(* Logix 5000 project; controller SX_V040001_C001 vendor 1 type 14 code 77 rev 16.23; software revision 16.04; part 21 of 35 *)
(* tags used below, declared in another part *)
   ALL_KINDS : INT[90];
   Basic : INT;
   G_DInput : DINT[3];
   G_DOutput : DINT[3];
   METERING : INT[44];
   METERING_PULSE : DINT[14];
   NOTDOS : INT[6];
   PARAMETER : INT[501];
(* MainProgram, continued *)

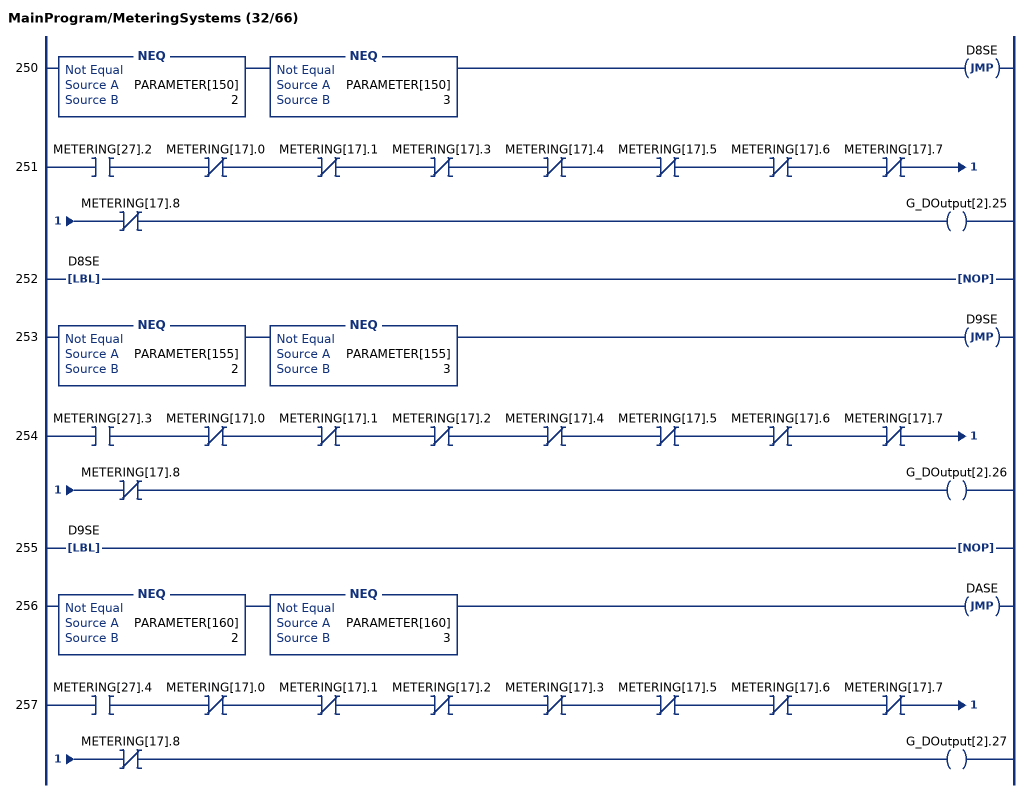
   [picture p456: MainProgram/MeteringSystems rungs 250-257]
   250: NEQ(PARAMETER[150],2)NEQ(PARAMETER[150],3)JMP(D8SE);
   251: XIC(METERING[27].2)XIO(METERING[17].0)XIO(METERING[17].1)XIO(METERING[17].3)XIO(METERING[17].4)XIO(METERING[17].5)XIO(METERING[17].6)XIO(METERING[17].7)XIO(METERING[17].8)OTE(G_DOutput[2].25);
   252: LBL(D8SE)NOP();
   253: NEQ(PARAMETER[155],2)NEQ(PARAMETER[155],3)JMP(D9SE);
   254: XIC(METERING[27].3)XIO(METERING[17].0)XIO(METERING[17].1)XIO(METERING[17].2)XIO(METERING[17].4)XIO(METERING[17].5)XIO(METERING[17].6)XIO(METERING[17].7)XIO(METERING[17].8)OTE(G_DOutput[2].26);
   255: LBL(D9SE)NOP();
   256: NEQ(PARAMETER[160],2)NEQ(PARAMETER[160],3)JMP(DASE);
   257: XIC(METERING[27].4)XIO(METERING[17].0)XIO(METERING[17].1)XIO(METERING[17].2)XIO(METERING[17].3)XIO(METERING[17].5)XIO(METERING[17].6)XIO(METERING[17].7)XIO(METERING[17].8)OTE(G_DOutput[2].27);
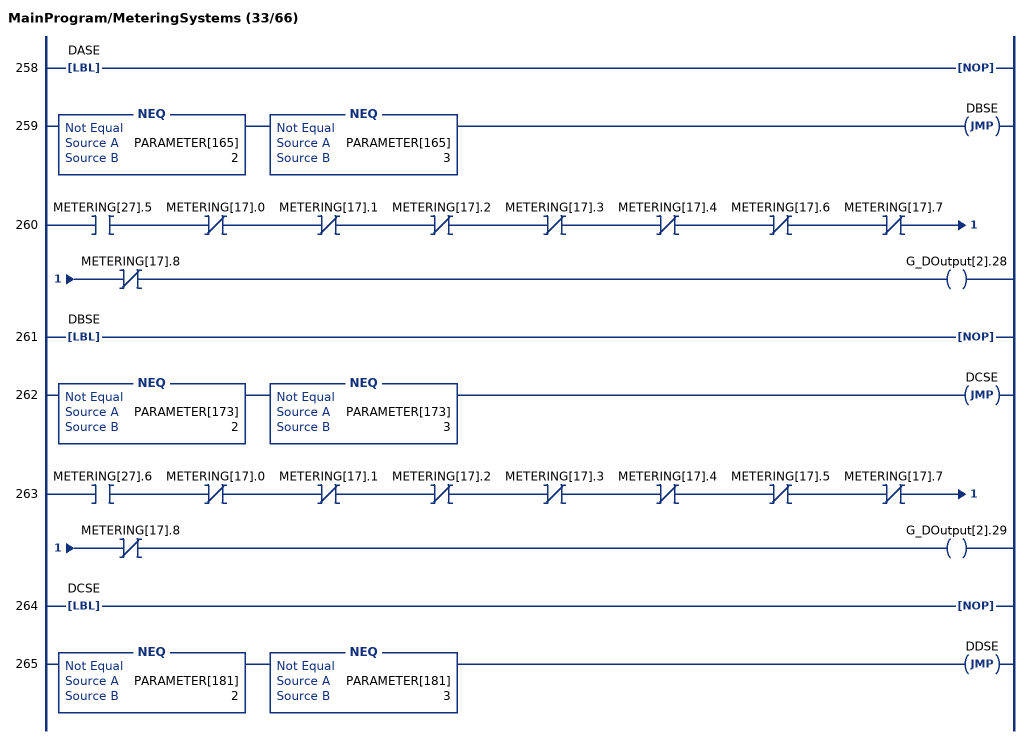
   258: LBL(DASE)NOP();
   259: NEQ(PARAMETER[165],2)NEQ(PARAMETER[165],3)JMP(DBSE);
   260: XIC(METERING[27].5)XIO(METERING[17].0)XIO(METERING[17].1)XIO(METERING[17].2)XIO(METERING[17].3)XIO(METERING[17].4)XIO(METERING[17].6)XIO(METERING[17].7)XIO(METERING[17].8)OTE(G_DOutput[2].28);
   261: LBL(DBSE)NOP();
   262: NEQ(PARAMETER[173],2)NEQ(PARAMETER[173],3)JMP(DCSE);
   263: XIC(METERING[27].6)XIO(METERING[17].0)XIO(METERING[17].1)XIO(METERING[17].2)XIO(METERING[17].3)XIO(METERING[17].4)XIO(METERING[17].5)XIO(METERING[17].7)XIO(METERING[17].8)OTE(G_DOutput[2].29);
   264: LBL(DCSE)NOP();
   265: NEQ(PARAMETER[181],2)NEQ(PARAMETER[181],3)JMP(DDSE);
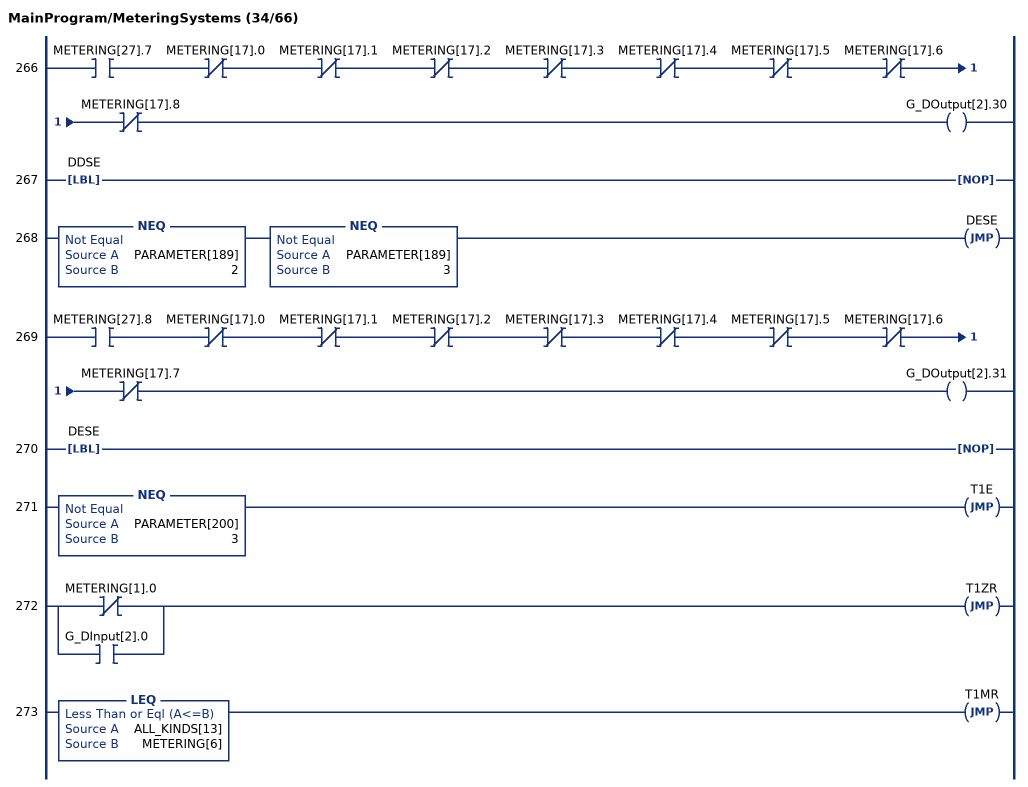
   266: XIC(METERING[27].7)XIO(METERING[17].0)XIO(METERING[17].1)XIO(METERING[17].2)XIO(METERING[17].3)XIO(METERING[17].4)XIO(METERING[17].5)XIO(METERING[17].6)XIO(METERING[17].8)OTE(G_DOutput[2].30);
   267: LBL(DDSE)NOP();
   268: NEQ(PARAMETER[189],2)NEQ(PARAMETER[189],3)JMP(DESE);
   269: XIC(METERING[27].8)XIO(METERING[17].0)XIO(METERING[17].1)XIO(METERING[17].2)XIO(METERING[17].3)XIO(METERING[17].4)XIO(METERING[17].5)XIO(METERING[17].6)XIO(METERING[17].7)OTE(G_DOutput[2].31);
   270: LBL(DESE)NOP();
   271: NEQ(PARAMETER[200],3)JMP(T1E);
   272: [XIO(METERING[1].0) ,XIC(G_DInput[2].0) ]JMP(T1ZR);
   273: LEQ(ALL_KINDS[13],METERING[6])JMP(T1MR);
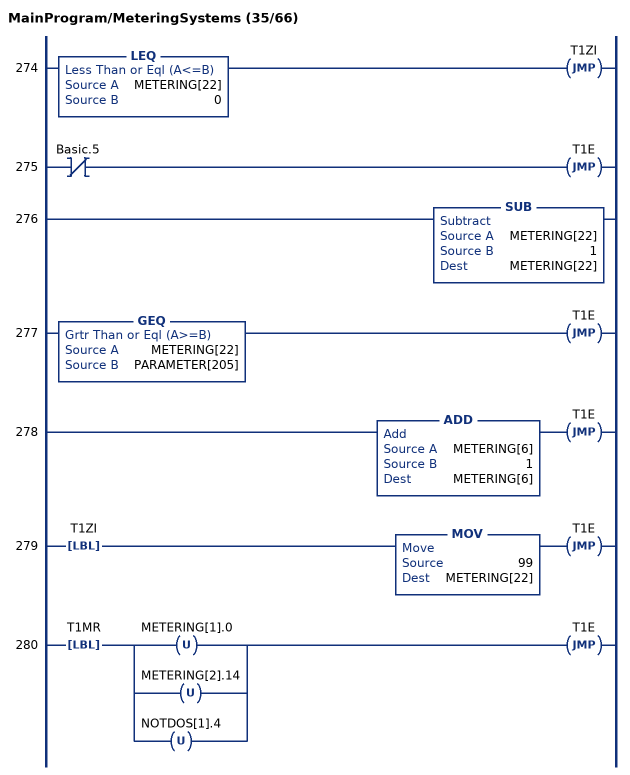
   274: LEQ(METERING[22],0)JMP(T1ZI);
   275: XIO(Basic.5)JMP(T1E);
   276: SUB(METERING[22],1,METERING[22]);
   277: GEQ(METERING[22],PARAMETER[205])JMP(T1E);
   278: ADD(METERING[6],1,METERING[6])JMP(T1E);
   279: LBL(T1ZI)MOV(99,METERING[22])JMP(T1E);
   280: LBL(T1MR)[OTU(METERING[1].0) ,OTU(METERING[2].14) ,OTU(NOTDOS[1].4) ]JMP(T1E);
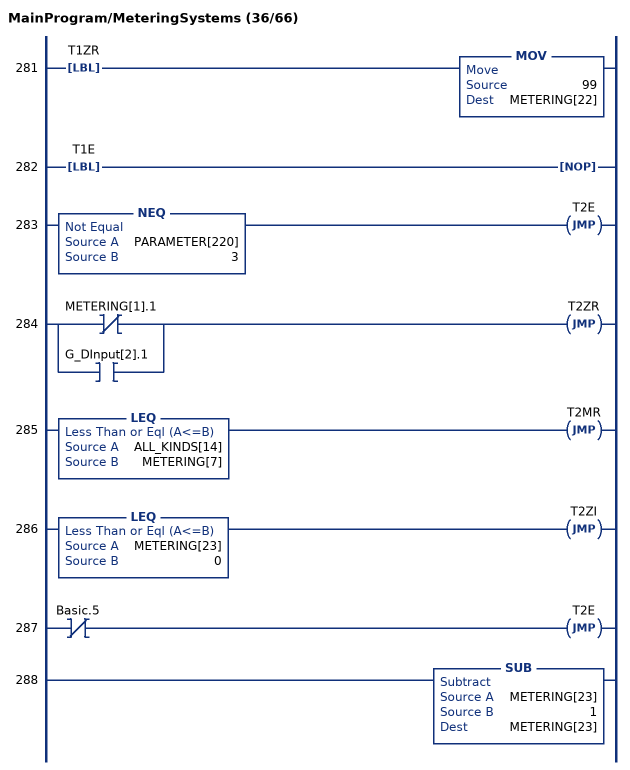
   281: LBL(T1ZR)MOV(99,METERING[22]);
   282: LBL(T1E)NOP();
   283: NEQ(PARAMETER[220],3)JMP(T2E);
   284: [XIO(METERING[1].1) ,XIC(G_DInput[2].1) ]JMP(T2ZR);
   285: LEQ(ALL_KINDS[14],METERING[7])JMP(T2MR);
   286: LEQ(METERING[23],0)JMP(T2ZI);
   287: XIO(Basic.5)JMP(T2E);
   288: SUB(METERING[23],1,METERING[23]);
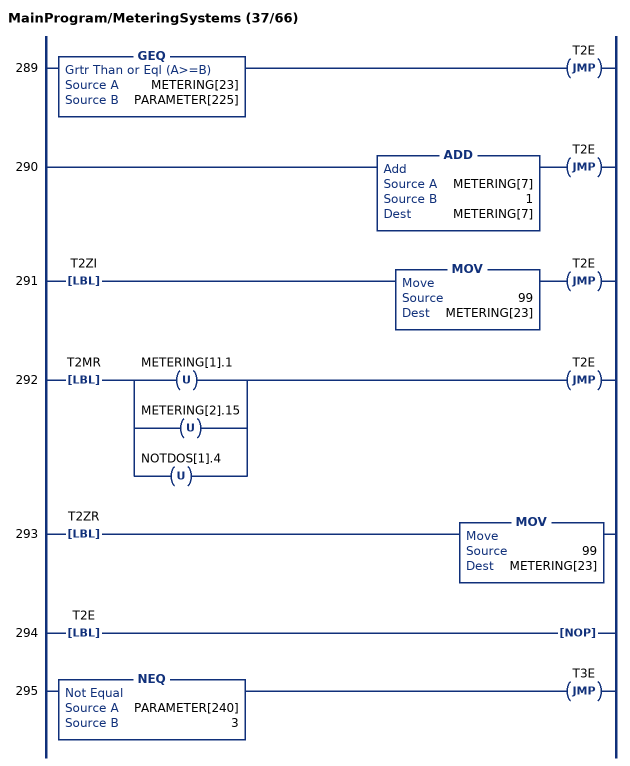
   289: GEQ(METERING[23],PARAMETER[225])JMP(T2E);
   290: ADD(METERING[7],1,METERING[7])JMP(T2E);
   291: LBL(T2ZI)MOV(99,METERING[23])JMP(T2E);
   292: LBL(T2MR)[OTU(METERING[1].1) ,OTU(METERING[2].15) ,OTU(NOTDOS[1].4) ]JMP(T2E);
   293: LBL(T2ZR)MOV(99,METERING[23]);
   294: LBL(T2E)NOP();
   295: NEQ(PARAMETER[240],3)JMP(T3E);
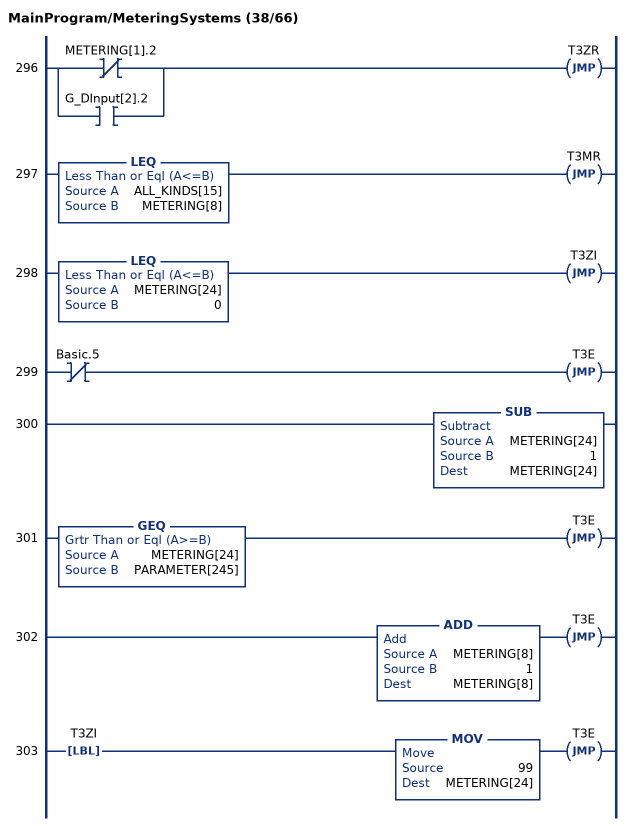
   296: [XIO(METERING[1].2) ,XIC(G_DInput[2].2) ]JMP(T3ZR);
   297: LEQ(ALL_KINDS[15],METERING[8])JMP(T3MR);
   298: LEQ(METERING[24],0)JMP(T3ZI);
   299: XIO(Basic.5)JMP(T3E);
   300: SUB(METERING[24],1,METERING[24]);
   301: GEQ(METERING[24],PARAMETER[245])JMP(T3E);
   302: ADD(METERING[8],1,METERING[8])JMP(T3E);
   303: LBL(T3ZI)MOV(99,METERING[24])JMP(T3E);
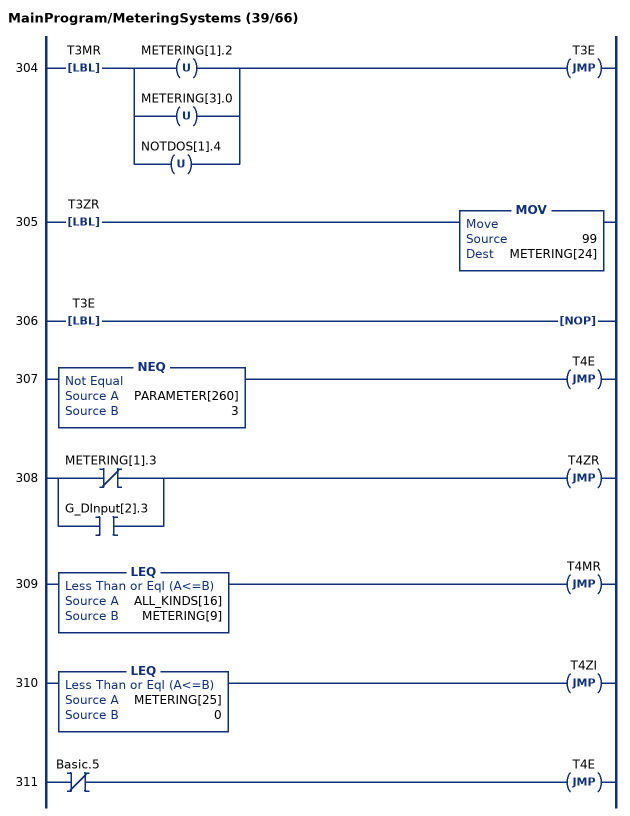
   304: LBL(T3MR)[OTU(METERING[1].2) ,OTU(METERING[3].0) ,OTU(NOTDOS[1].4) ]JMP(T3E);
   305: LBL(T3ZR)MOV(99,METERING[24]);
   306: LBL(T3E)NOP();
   307: NEQ(PARAMETER[260],3)JMP(T4E);
   308: [XIO(METERING[1].3) ,XIC(G_DInput[2].3) ]JMP(T4ZR);
   309: LEQ(ALL_KINDS[16],METERING[9])JMP(T4MR);
   310: LEQ(METERING[25],0)JMP(T4ZI);
   311: XIO(Basic.5)JMP(T4E);
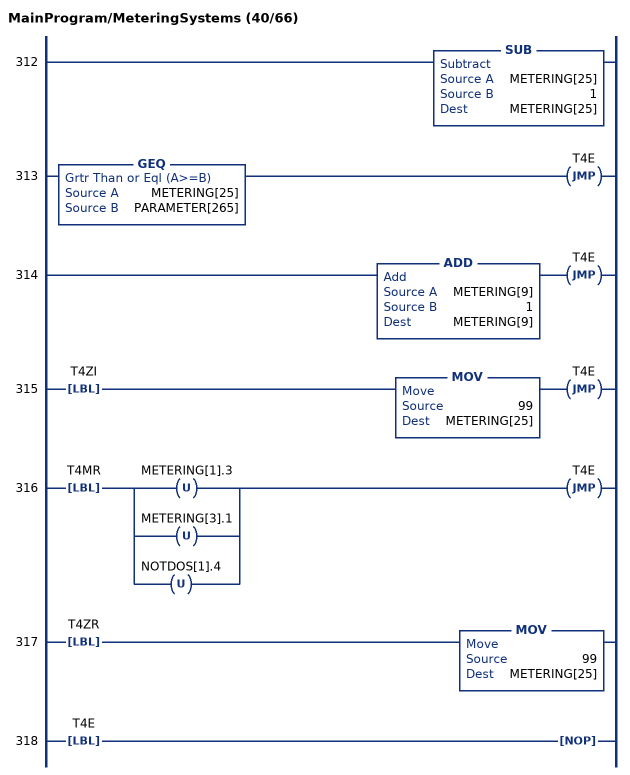
   312: SUB(METERING[25],1,METERING[25]);
   313: GEQ(METERING[25],PARAMETER[265])JMP(T4E);
   314: ADD(METERING[9],1,METERING[9])JMP(T4E);
   315: LBL(T4ZI)MOV(99,METERING[25])JMP(T4E);
   316: LBL(T4MR)[OTU(METERING[1].3) ,OTU(METERING[3].1) ,OTU(NOTDOS[1].4) ]JMP(T4E);
   317: LBL(T4ZR)MOV(99,METERING[25]);
   318: LBL(T4E)NOP();
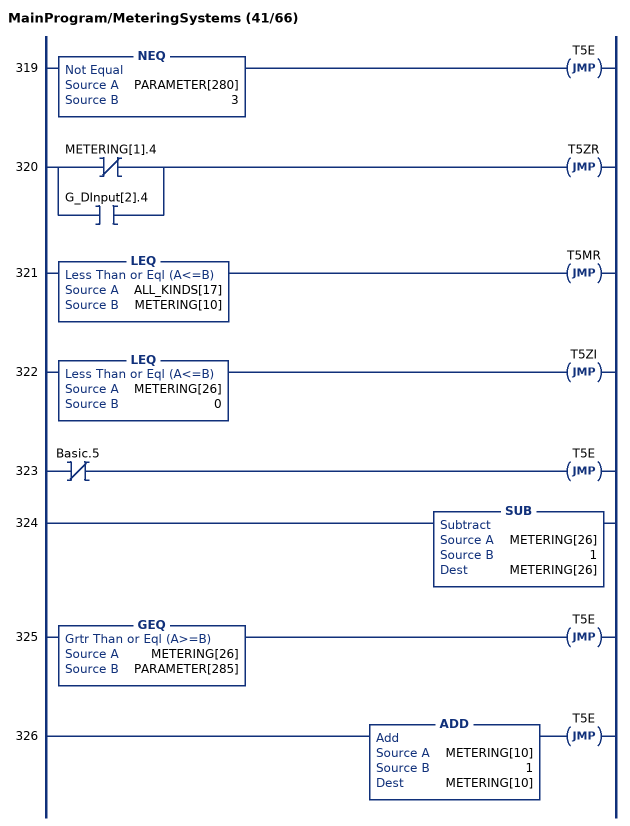
   319: NEQ(PARAMETER[280],3)JMP(T5E);
   320: [XIO(METERING[1].4) ,XIC(G_DInput[2].4) ]JMP(T5ZR);
   321: LEQ(ALL_KINDS[17],METERING[10])JMP(T5MR);
   322: LEQ(METERING[26],0)JMP(T5ZI);
   323: XIO(Basic.5)JMP(T5E);
   324: SUB(METERING[26],1,METERING[26]);
   325: GEQ(METERING[26],PARAMETER[285])JMP(T5E);
   326: ADD(METERING[10],1,METERING[10])JMP(T5E);
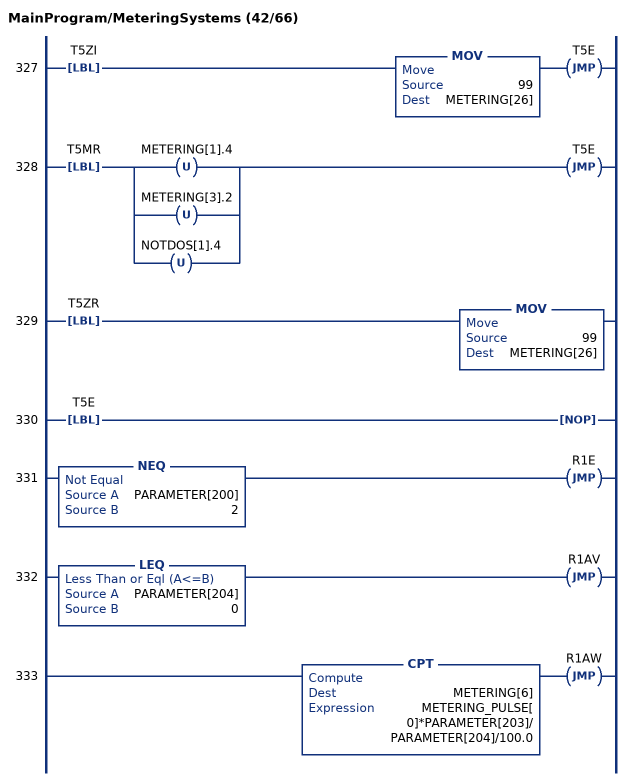
   327: LBL(T5ZI)MOV(99,METERING[26])JMP(T5E);
   328: LBL(T5MR)[OTU(METERING[1].4) ,OTU(METERING[3].2) ,OTU(NOTDOS[1].4) ]JMP(T5E);
   329: LBL(T5ZR)MOV(99,METERING[26]);
   330: LBL(T5E)NOP();
   331: NEQ(PARAMETER[200],2)JMP(R1E);
   332: LEQ(PARAMETER[204],0)JMP(R1AV);
   333: CPT(METERING[6],METERING_PULSE[0]*PARAMETER[203]/PARAMETER[204]/100.0)JMP(R1AW);
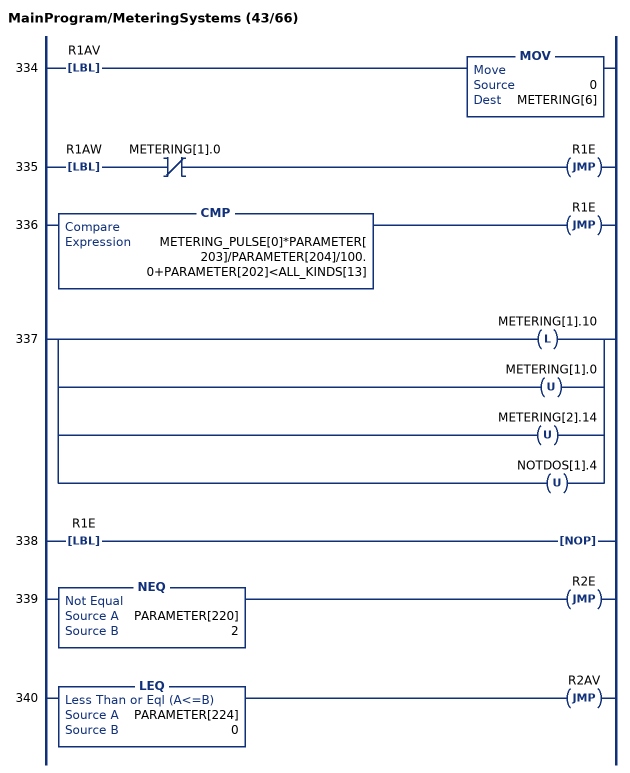
   334: LBL(R1AV)MOV(0,METERING[6]);
   335: LBL(R1AW)XIO(METERING[1].0)JMP(R1E);
   336: CMP(METERING_PULSE[0]*PARAMETER[203]/PARAMETER[204]/100.0+PARAMETER[202]<ALL_KINDS[13])JMP(R1E);
   337: [OTL(METERING[1].10) ,OTU(METERING[1].0) ,OTU(METERING[2].14) ,OTU(NOTDOS[1].4) ];
   338: LBL(R1E)NOP();
   339: NEQ(PARAMETER[220],2)JMP(R2E);
   340: LEQ(PARAMETER[224],0)JMP(R2AV);
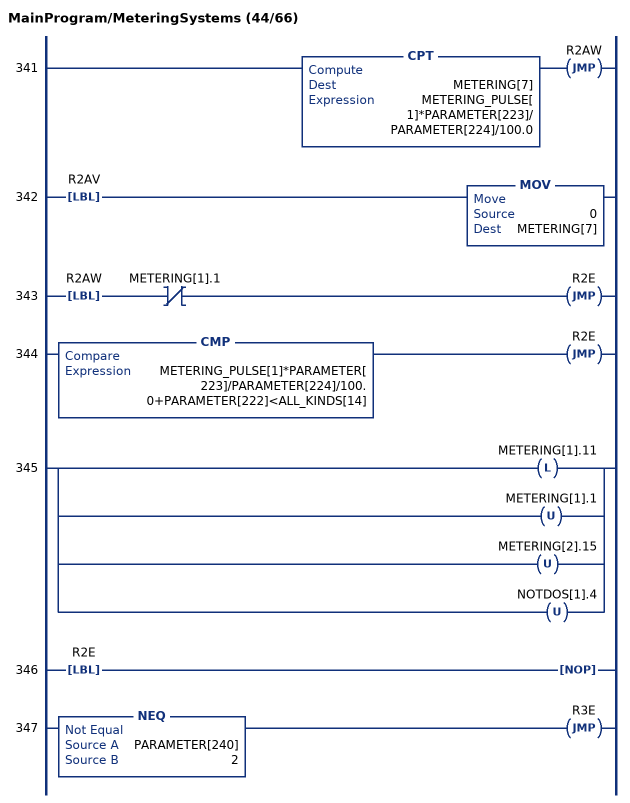
   341: CPT(METERING[7],METERING_PULSE[1]*PARAMETER[223]/PARAMETER[224]/100.0)JMP(R2AW);
   342: LBL(R2AV)MOV(0,METERING[7]);
   343: LBL(R2AW)XIO(METERING[1].1)JMP(R2E);
   344: CMP(METERING_PULSE[1]*PARAMETER[223]/PARAMETER[224]/100.0+PARAMETER[222]<ALL_KINDS[14])JMP(R2E);
   345: [OTL(METERING[1].11) ,OTU(METERING[1].1) ,OTU(METERING[2].15) ,OTU(NOTDOS[1].4) ];
   346: LBL(R2E)NOP();
   347: NEQ(PARAMETER[240],2)JMP(R3E);
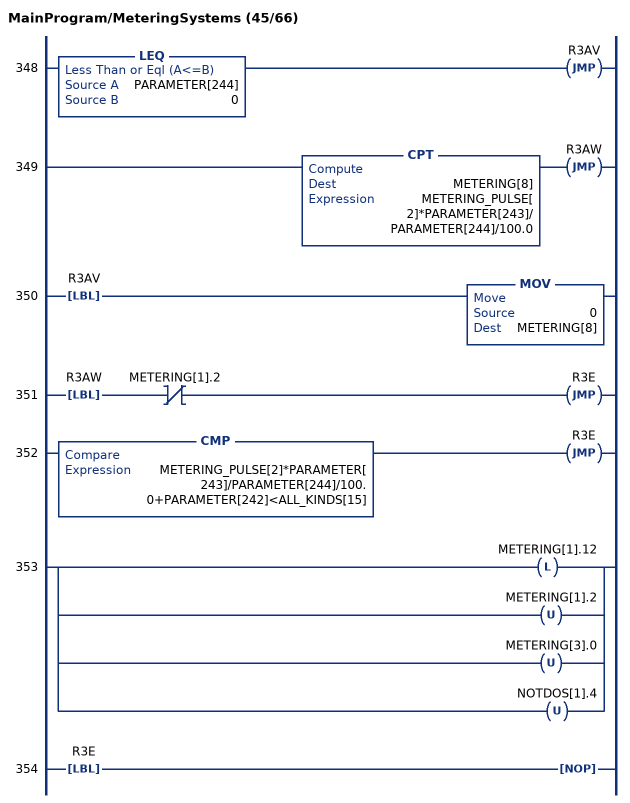
   348: LEQ(PARAMETER[244],0)JMP(R3AV);
   349: CPT(METERING[8],METERING_PULSE[2]*PARAMETER[243]/PARAMETER[244]/100.0)JMP(R3AW);
   350: LBL(R3AV)MOV(0,METERING[8]);
   351: LBL(R3AW)XIO(METERING[1].2)JMP(R3E);
   352: CMP(METERING_PULSE[2]*PARAMETER[243]/PARAMETER[244]/100.0+PARAMETER[242]<ALL_KINDS[15])JMP(R3E);
   353: [OTL(METERING[1].12) ,OTU(METERING[1].2) ,OTU(METERING[3].0) ,OTU(NOTDOS[1].4) ];
   354: LBL(R3E)NOP();
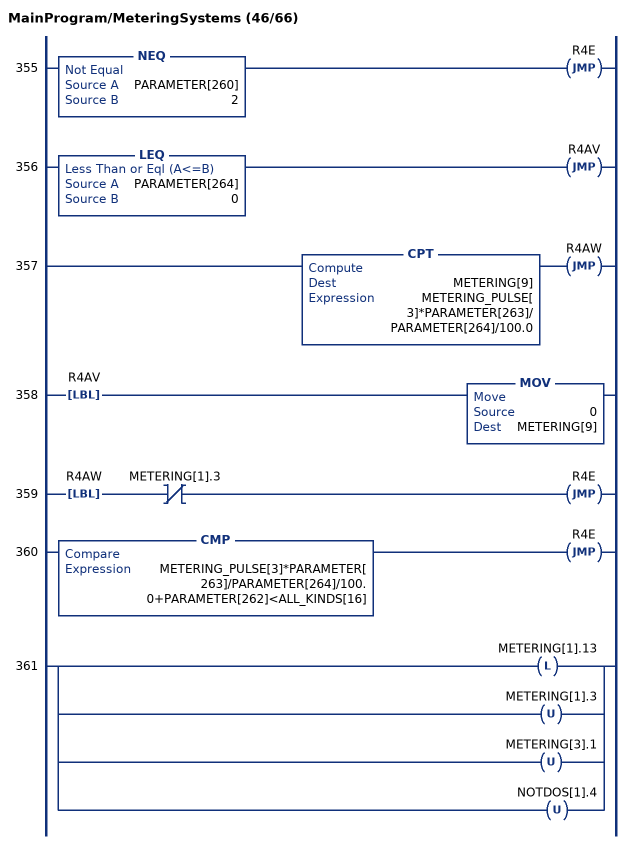
   355: NEQ(PARAMETER[260],2)JMP(R4E);
   356: LEQ(PARAMETER[264],0)JMP(R4AV);
   357: CPT(METERING[9],METERING_PULSE[3]*PARAMETER[263]/PARAMETER[264]/100.0)JMP(R4AW);
   358: LBL(R4AV)MOV(0,METERING[9]);
   359: LBL(R4AW)XIO(METERING[1].3)JMP(R4E);
   360: CMP(METERING_PULSE[3]*PARAMETER[263]/PARAMETER[264]/100.0+PARAMETER[262]<ALL_KINDS[16])JMP(R4E);
   361: [OTL(METERING[1].13) ,OTU(METERING[1].3) ,OTU(METERING[3].1) ,OTU(NOTDOS[1].4) ];
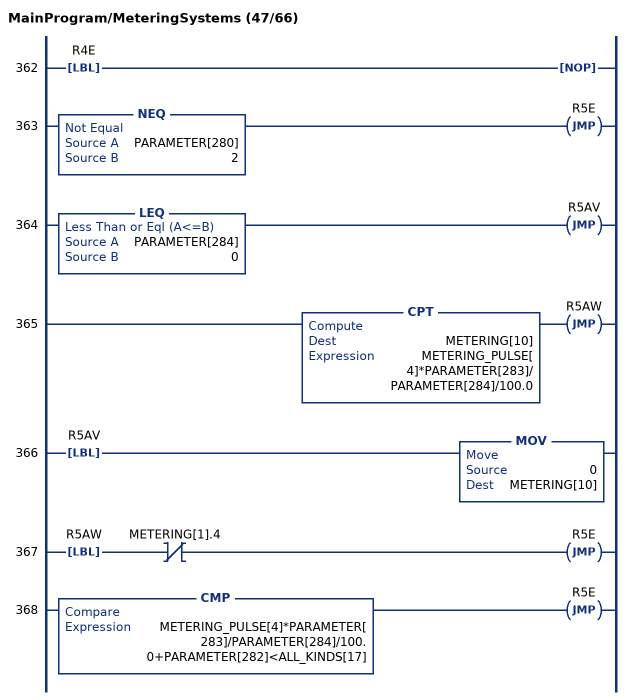
   362: LBL(R4E)NOP();
   363: NEQ(PARAMETER[280],2)JMP(R5E);
   364: LEQ(PARAMETER[284],0)JMP(R5AV);
   365: CPT(METERING[10],METERING_PULSE[4]*PARAMETER[283]/PARAMETER[284]/100.0)JMP(R5AW);
   366: LBL(R5AV)MOV(0,METERING[10]);
   367: LBL(R5AW)XIO(METERING[1].4)JMP(R5E);
   368: CMP(METERING_PULSE[4]*PARAMETER[283]/PARAMETER[284]/100.0+PARAMETER[282]<ALL_KINDS[17])JMP(R5E);
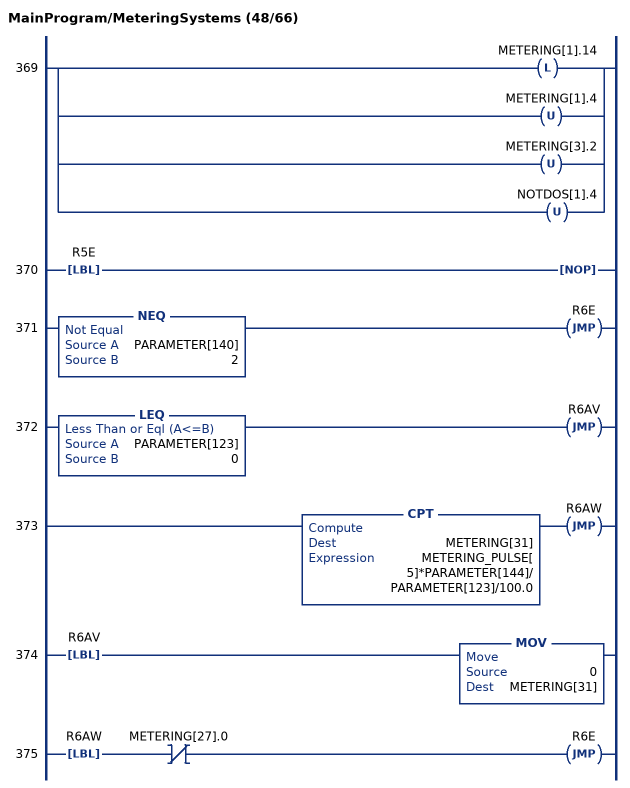
   369: [OTL(METERING[1].14) ,OTU(METERING[1].4) ,OTU(METERING[3].2) ,OTU(NOTDOS[1].4) ];
   370: LBL(R5E)NOP();
   371: NEQ(PARAMETER[140],2)JMP(R6E);
   372: LEQ(PARAMETER[123],0)JMP(R6AV);
   373: CPT(METERING[31],METERING_PULSE[5]*PARAMETER[144]/PARAMETER[123]/100.0)JMP(R6AW);
   374: LBL(R6AV)MOV(0,METERING[31]);
   375: LBL(R6AW)XIO(METERING[27].0)JMP(R6E);
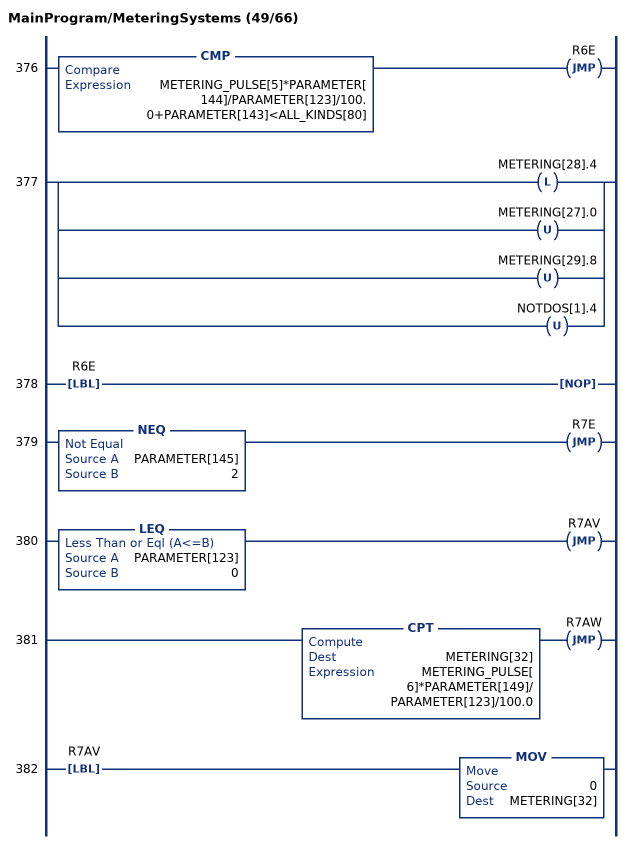
   376: CMP(METERING_PULSE[5]*PARAMETER[144]/PARAMETER[123]/100.0+PARAMETER[143]<ALL_KINDS[80])JMP(R6E);
   377: [OTL(METERING[28].4) ,OTU(METERING[27].0) ,OTU(METERING[29].8) ,OTU(NOTDOS[1].4) ];
   378: LBL(R6E)NOP();
   379: NEQ(PARAMETER[145],2)JMP(R7E);
   380: LEQ(PARAMETER[123],0)JMP(R7AV);
   381: CPT(METERING[32],METERING_PULSE[6]*PARAMETER[149]/PARAMETER[123]/100.0)JMP(R7AW);
   382: LBL(R7AV)MOV(0,METERING[32]);
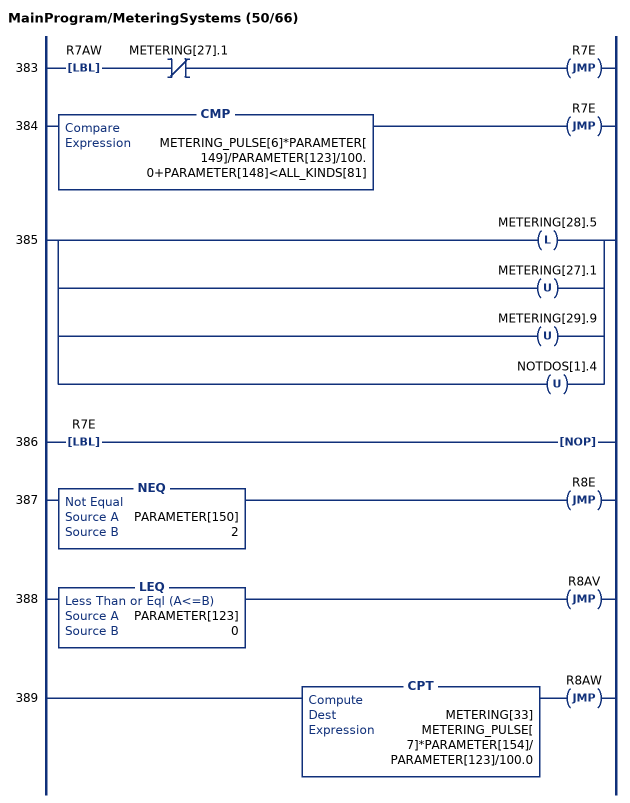
   383: LBL(R7AW)XIO(METERING[27].1)JMP(R7E);
   384: CMP(METERING_PULSE[6]*PARAMETER[149]/PARAMETER[123]/100.0+PARAMETER[148]<ALL_KINDS[81])JMP(R7E);
   385: [OTL(METERING[28].5) ,OTU(METERING[27].1) ,OTU(METERING[29].9) ,OTU(NOTDOS[1].4) ];
   386: LBL(R7E)NOP();
   387: NEQ(PARAMETER[150],2)JMP(R8E);
   388: LEQ(PARAMETER[123],0)JMP(R8AV);
   389: CPT(METERING[33],METERING_PULSE[7]*PARAMETER[154]/PARAMETER[123]/100.0)JMP(R8AW);
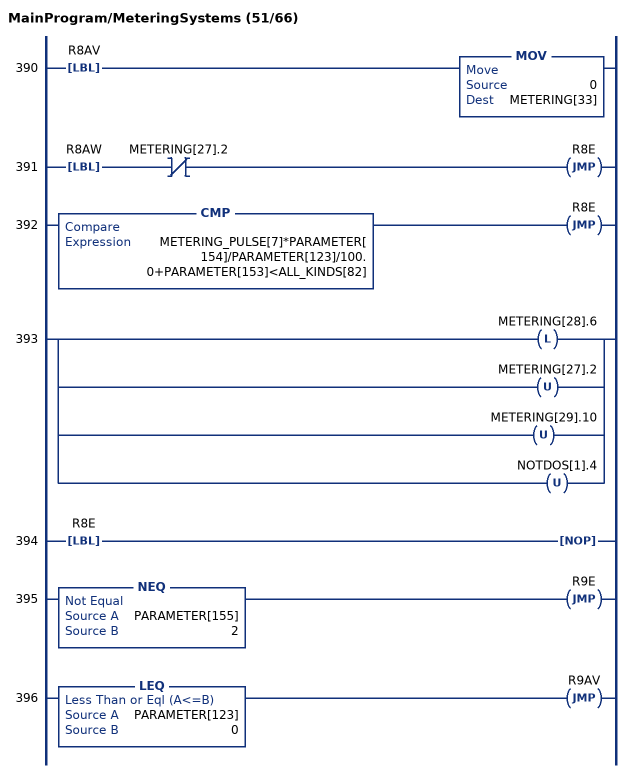
   390: LBL(R8AV)MOV(0,METERING[33]);
   391: LBL(R8AW)XIO(METERING[27].2)JMP(R8E);
   392: CMP(METERING_PULSE[7]*PARAMETER[154]/PARAMETER[123]/100.0+PARAMETER[153]<ALL_KINDS[82])JMP(R8E);
   393: [OTL(METERING[28].6) ,OTU(METERING[27].2) ,OTU(METERING[29].10) ,OTU(NOTDOS[1].4) ];
   394: LBL(R8E)NOP();
   395: NEQ(PARAMETER[155],2)JMP(R9E);
   396: LEQ(PARAMETER[123],0)JMP(R9AV);
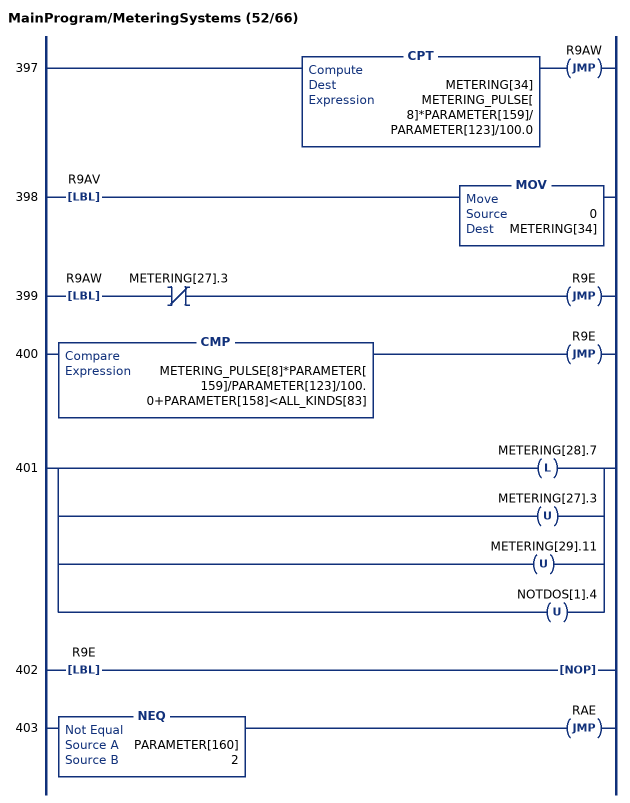
   397: CPT(METERING[34],METERING_PULSE[8]*PARAMETER[159]/PARAMETER[123]/100.0)JMP(R9AW);
   398: LBL(R9AV)MOV(0,METERING[34]);
   399: LBL(R9AW)XIO(METERING[27].3)JMP(R9E);
   400: CMP(METERING_PULSE[8]*PARAMETER[159]/PARAMETER[123]/100.0+PARAMETER[158]<ALL_KINDS[83])JMP(R9E);
   401: [OTL(METERING[28].7) ,OTU(METERING[27].3) ,OTU(METERING[29].11) ,OTU(NOTDOS[1].4) ];
   402: LBL(R9E)NOP();
   403: NEQ(PARAMETER[160],2)JMP(RAE);
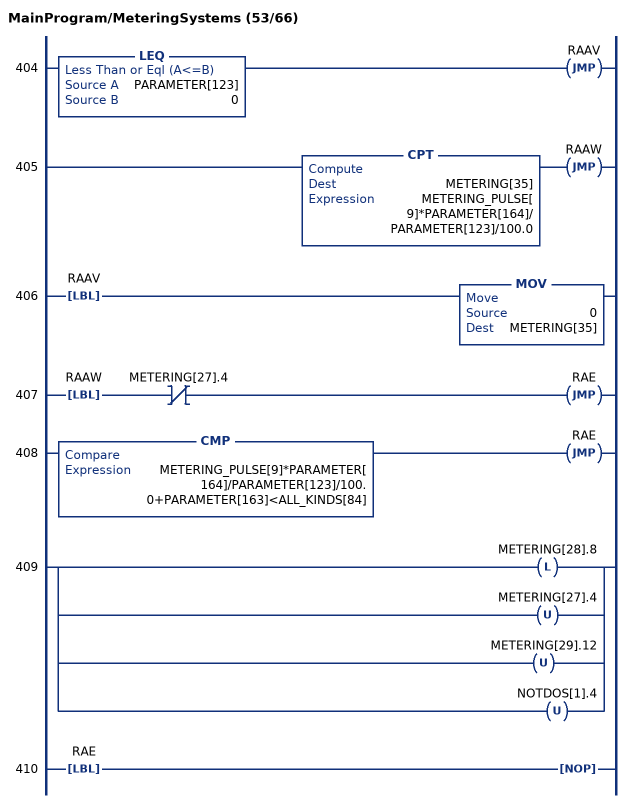
   404: LEQ(PARAMETER[123],0)JMP(RAAV);
   405: CPT(METERING[35],METERING_PULSE[9]*PARAMETER[164]/PARAMETER[123]/100.0)JMP(RAAW);
   406: LBL(RAAV)MOV(0,METERING[35]);
   407: LBL(RAAW)XIO(METERING[27].4)JMP(RAE);
   408: CMP(METERING_PULSE[9]*PARAMETER[164]/PARAMETER[123]/100.0+PARAMETER[163]<ALL_KINDS[84])JMP(RAE);
   409: [OTL(METERING[28].8) ,OTU(METERING[27].4) ,OTU(METERING[29].12) ,OTU(NOTDOS[1].4) ];
   410: LBL(RAE)NOP();
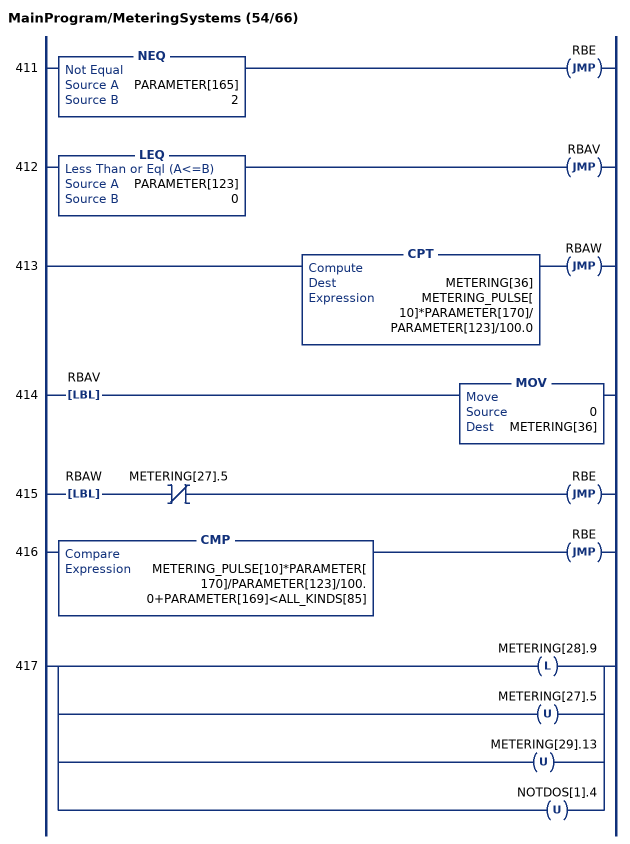
   411: NEQ(PARAMETER[165],2)JMP(RBE);
   412: LEQ(PARAMETER[123],0)JMP(RBAV);
   413: CPT(METERING[36],METERING_PULSE[10]*PARAMETER[170]/PARAMETER[123]/100.0)JMP(RBAW);
   414: LBL(RBAV)MOV(0,METERING[36]);
   415: LBL(RBAW)XIO(METERING[27].5)JMP(RBE);
   416: CMP(METERING_PULSE[10]*PARAMETER[170]/PARAMETER[123]/100.0+PARAMETER[169]<ALL_KINDS[85])JMP(RBE);
   417: [OTL(METERING[28].9) ,OTU(METERING[27].5) ,OTU(METERING[29].13) ,OTU(NOTDOS[1].4) ];
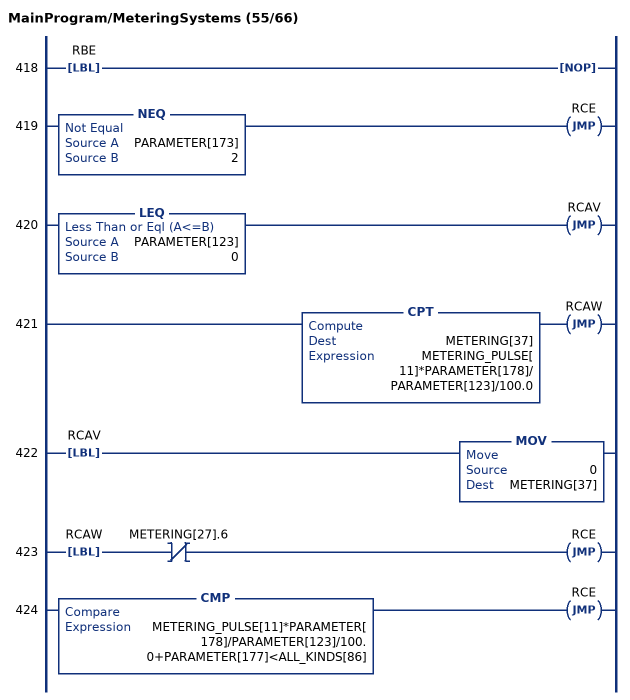
   418: LBL(RBE)NOP();
   419: NEQ(PARAMETER[173],2)JMP(RCE);
   420: LEQ(PARAMETER[123],0)JMP(RCAV);
   421: CPT(METERING[37],METERING_PULSE[11]*PARAMETER[178]/PARAMETER[123]/100.0)JMP(RCAW);
   422: LBL(RCAV)MOV(0,METERING[37]);
   423: LBL(RCAW)XIO(METERING[27].6)JMP(RCE);
   424: CMP(METERING_PULSE[11]*PARAMETER[178]/PARAMETER[123]/100.0+PARAMETER[177]<ALL_KINDS[86])JMP(RCE);
